FUNCTION_BLOCK FB_CalculateXrayAbsorptionConstant_Test EXTENDS TcUnit.FB_TestSuite
VAR
END_VAR


GivenValidInputsExpectCorrectResult();


METHOD PRIVATE GivenValidInputsExpectCorrectResult
VAR
    fResult : LREAL;
END_VAR

TEST('GivenValidInputsExpectCorrectResult');

fResult := F_CalculateXrayAbsorptionConstant(
    f2 := 0.0058932368755846573,
    fPhotonEnergy_eV := 10000,
    fDensity_gm3 := 3.51e6,
    fAtomicWeight := 12.0107
);

AssertEquals_LREAL(
    Expected := 724.7224642932565,
    Actual := fResult,
    Delta := 1e-9,
    Message := 'Incorrect result.'
);

TEST_FINISHED();
END_METHOD

END_FUNCTION_BLOCK

(* stored: Version 1.1.0.1
   POU FB_CalculateXrayAbsorptionConstant_Test: Id {1105c2f4-4390-4877-9b15-5c2eb2769fd4}, SpecialFunc None
   Method GivenValidInputsExpectCorrectResult: Id {fd44bfc3-64a1-4410-9d8e-17840a50d078} *)
